TYPE DUT_ResourcesByType :
STRUCT
	return_value	: DINT;
	ReaourceType	: STRING(50);
END_STRUCT
END_TYPE

(* stored: Version 1.1.0.1, ProductVersion 3.1.4024.15
   DUT DUT_ResourcesByType: Id {69d79b6b-9135-47c5-9202-79ab8903b45f} *)
